(* IEC 61131-3 sources: programs/VI-54/VI-54_20171205/VI-54_20171205/Stations/Screen/LseClass170718/Class/Comm_RecvData, 1 file *)

(* ---- Comm_RecvData.st ---- *)
(*!
<Class
	Name               = "Comm_RecvData"
	Revision           = "0.4"
	RealtimeTask       = "false"
	CyclicTask         = "false"
	BackgroundTask     = "false"
	Sigmatek           = "false"
	OSInterface        = "false"
	HighPriority       = "false"
	Automatic          = "false"
	UpdateMode         = "Prescan"
	SharedCommandTable = "true"
	Objectsize         = "(600,240)"
	Comment            = "Receiving data via communication class.">
	<Channels>
		<Server Name="ClassSvr" Visualized="false" Initialize="false" WriteProtected="true" Retentive="false"/>
		<Server Name="sMyID" Visualized="false" Initialize="true" WriteProtected="true" Retentive="false" Comment="Source communication id number."/>
		<Server Name="sRecvCnt" Visualized="false" Initialize="false" WriteProtected="false" Retentive="false" Comment="Counter for received data blocks."/>
		<Client Name="cDataMng" Required="true" Internal="false" Comment="Connection to communication data manager."/>
	</Channels>
	<RevDoku>
		<Owner/>
		<Dokumentation Revision="0.4" Date="2014-12-02" Author="hötant" Company="DETS" Description="changed init methode ( _firstscan is too late )"/>
		<Dokumentation Revision="0.3" Date="2014-11-11" Author="hötant" Company="DETS" Description="added new methode CallBackReciverCMD"/>
		<Dokumentation Revision="0.2" Date="2014-10-22" Author="hötant" Company="DETS" Description="added new output parameter to  method CallBackReciver"/>
		<Dokumentation Revision="0.1" Date="2014-10-21" Author="SJO" Company="DETS" Description="SJO_09102014 added Background method"/>
	</RevDoku>
</Class>
*)
Comm_RecvData : CLASS
  //Servers:
	ClassSvr 	: SvrChCmd_DINT;
	sMyID 	: SvrCh_DINT;
	sRecvCnt 	: SvrCh_DINT;
  //Clients:
	cDataMng 	: CltChCmd_DataManager;
  //Variables:
		InitCounter 	: DINT;
  //Functions:

	FUNCTION VIRTUAL GLOBAL Init;

	FUNCTION VIRTUAL GLOBAL CallBackReciver
		VAR_INPUT
			DestinationID 	: DINT;
			SourceID 	: DINT;
			size 	: UDINT;
			pdata 	: ^USINT;
		END_VAR
		VAR_OUTPUT
			retcode 	: BOOL;			//! <Variable Comment="TRUE .. erfolgreich Empfangen .._MNG_Recived &#13;&#10;FALSE.. Fehler beim Empfangen .._MNG_GlobalReciveError" Name="CallBackReciver.retcode"/>
		END_VAR;

	FUNCTION VIRTUAL GLOBAL CallBackReciverCMD
		VAR_INPUT
			DestinationID 	: DINT;
			SourceID 	: DINT;
			size 	: UDINT;
			pdata 	: ^USINT;
			OptCMD 	: USINT;
		END_VAR
		VAR_OUTPUT
			retcode 	: BOOL;
		END_VAR;
  //Tables:
	FUNCTION @STD
		VAR_OUTPUT
			ret_code	: CONFSTATES;
		END_VAR;
	FUNCTION GLOBAL TAB @CT_;
END_CLASS;

#pragma usingLtd DataManager

FUNCTION GLOBAL Comm_RecvData_CB
	VAR_INPUT
		pthis 	: ^void;
		DestinationID 	: DINT;
		SourceID 	: DINT;
		size 	: UDINT;
		pdata 	: ^USINT;
	END_VAR
  var_output
    retcode : bool;
  end_var

  retcode := pthis$^Comm_RecvData^.CallBackReciver(DestinationID, SourceID, size, pdata);
  pthis$^Comm_RecvData^.sRecvCnt +=1;

END_FUNCTION

#pragma warning(disable:73);
FUNCTION VIRTUAL GLOBAL Comm_RecvData::CallBackReciver
	VAR_INPUT
		DestinationID 	: DINT;
		SourceID 	: DINT;
		size 	: UDINT;
		pdata 	: ^USINT;
	END_VAR
	VAR_OUTPUT
		retcode 	: BOOL;
	END_VAR

  retcode := CallBackReciverCMD(DestinationID:=(DestinationID AND 16#00FFFFFF),
                                SourceID:=SourceID,
                                size:=size,
                                pdata:=pdata,
                                OptCMD:= to_usint((DestinationID$udint AND 16#FF000000) shr 24)  );

END_FUNCTION
#pragma warning(default:73);

#pragma warning(disable:73);
FUNCTION VIRTUAL GLOBAL Comm_RecvData::CallBackReciverCMD
	VAR_INPUT
		DestinationID 	: DINT;
		SourceID 	: DINT;
		size 	: UDINT;
		pdata 	: ^USINT;
    OptCMD  : USINT;
	END_VAR
	VAR_OUTPUT
		retcode 	: BOOL;
	END_VAR

  // Daten wurden erfolgreich empfangen.
  retcode := TRUE;

END_FUNCTION
#pragma warning(default:73);

FUNCTION VIRTUAL GLOBAL Comm_RecvData::Init

  if InitCounter = 8 then
    cDataMng.ConnectReciver(udID:=sMyID, pThis:=this, pCallback:=#Comm_RecvData_CB());
  end_if;
  InitCounter +=1;

END_FUNCTION
